{attribute 'qualified_only'}
{attribute 'strict'}
TYPE ePOUState :
(
	OFF := 0,
	PowerUp := 1,
	Init := 2,
	Normal	:=	3,
	EMSTOP	:=	4,
	Shutdown := 5
);
END_TYPE

(* stored: Version 1.1.0.1, ProductVersion 3.1.4024.12
   DUT ePOUState: Id {b35bbe34-db77-4299-b7a1-58508a29fb67} *)
